  rq_init_comm_if_connected(9, "1")
  rq_init_comm_if_connected(2, "2")
  rq_init_comm_if_connected(3, "3")
  rq_init_comm_if_connected(4, "4")
  rq_print_connected_grippers()
  rq_gripper_communication_thread = run rq_gripper_communication()
  set_closed_norm(100.0, 1)
  set_open_norm(0.0, 1)
  set_closed_mm(0.0, 1)
  set_open_mm(50.0, 1)
  set_closed_norm(89.80392156862744, 2)
  set_open_norm(1.1764705882352942, 2)
  set_closed_mm(0.0, 2)
  set_open_mm(85.0, 2)
  set_closed_norm(100.0, 3)
  set_open_norm(0.0, 3)
  set_closed_mm(0.0, 3)
  set_open_mm(50.0, 3)
  set_closed_norm(100.0, 4)
  set_open_norm(0.0, 4)
  set_closed_mm(0.0, 4)
  set_open_mm(50.0, 4)
  rq_current_limit_enabled = False
  while(not rq_gripper_communication_thread_started):
      sleep(0.008)
  end
  # end: URCap Installation Node
  global Waypoint_1_p=p[.239154028168, -.112421187536, .388460805492, -2.190061121647, 2.239885105363, -.031522131746]
  global Waypoint_1_q=[0.08494941145181656, -1.356790379886963, -1.3501760959625244, 4.298311873073242, 1.5503448247909546, -12.457233563551696]
  global Waypoint_2_p=p[.353622143993, -.121329124968, .189938870353, -2.206384372041, 2.219086090555, -.015107570982]
  global Waypoint_2_q=[0.029603084549307823, -1.8911191425719203, -1.7472671270370483, 5.225752520352163, 1.5633039474487305, -12.537665781119856]
  global Waypoint_3_p=p[.353631843850, -.121307264267, .374404133955, -2.206378505151, 2.218976644385, -.015136018793]
  global Waypoint_3_q=[0.028919491916894913, -1.8426815472044886, -0.9176297783851624, 4.347720308894775, 1.5626927614212036, -12.531363688895496]
  global Waypoint_4_p=p[.353652148585, -.121293807225, .374372255201, -3.125989777988, .006696998981, .003111919112]
  global Waypoint_4_q=[0.02515784278512001, -1.855485578576559, -0.8932921886444092, 4.319008513087891, 1.5770167112350464, -14.107108545287538]
  global Waypoint_5_p=p[.363758828354, -.279187005666, .088904998077, -1.864461804969, .039872112715, .023313168997]
  global Waypoint_5_q=[-0.5345833937274378, -3.078116556207174, 0.038124863301412404, 3.5885044771381835, 2.5377118587493896, -15.200349044783998]
  global Waypoint_6_p=p[.362697799110, -.116842031967, .196258778113, -2.190025675108, 2.239949259838, -.031496290672]
  global Waypoint_6_q=[0.04410656914114952, -1.9051410160460414, -1.6960663795471191, 5.193034875183859, 1.5527570247650146, -12.506267488488945]
  global Waypoint_7_p=p[.362692894564, -.116852534259, .196244574783, -2.259726483789, -2.172286107875, .033806793645]
  global Waypoint_7_q=[0.04398636892437935, -1.9128123722472132, -1.6671544313430786, 5.131094622402944, 1.5524976253509521, -9.347179301569255]
  global Waypoint_8_p=p[.364841512775, -.116912589132, .188280404566, -3.140213348041, .061797284546, .022617550423]
  global Waypoint_8_q=[0.04088902473449707, -1.9356409511961878, -1.678733229637146, 5.171853232174673, 1.5633610486984253, -14.06320519445746]
  global Waypoint_9_p=p[.364848248729, -.116916737546, .353527898805, -3.140241647694, .061909886054, .022584279111]
  global Waypoint_9_q=[0.040220536291599274, -1.8723865948119105, -0.9687836766242981, 4.39864365636792, 1.5626797676086426, -14.057535123809267]
  global Waypoint_10_p=p[.360930807194, -.273182609942, .095849475862, -1.840638665045, .023655413076, -.007249116988]
  global Waypoint_10_q=[-0.5289800802813929, -2.9153500996031703, -0.2807917296886444, 3.7200543123432617, 2.5632033348083496, -15.246222686751771]
  global Waypoint_11_p=p[.358486190954, -.117341083615, .189882871874, -2.190038242218, 2.239881886121, -.031548557662]
  global Waypoint_11_q=[0.04321024566888809, -1.9022838077940882, -1.7338793277740479, 5.228053617268362, 1.5529053211212158, -12.50744832355717]
  global Waypoint_12_p=p[.358488238407, -.117335044807, .416524833090, -2.189975558032, 2.239914270517, -.031549652988]
  global Waypoint_12_q=[0.041965365409851074, -1.9908906422057093, -0.4767185151576996, 4.059401198024414, 1.5538296699523926, -12.499717981109413]
  global Waypoint_13_p=p[.358499834191, -.117338038000, .416498790970, -.024529661157, -3.133343015716, .032078362261]
  global Waypoint_13_q=[0.04467107728123665, -2.0224882564940394, -0.4105936884880066, 3.9957544046589355, 1.5432183742523193, -10.932522662470134]
  global Waypoint_14_p=p[.366071635210, -.114893443374, .213688173446, -.024436496176, -3.133440569951, .032084448400]
  global Waypoint_14_q=[0.05177054554224014, -1.8911673031248988, -1.61358642578125, 5.067582773953237, 1.5413740873336792, -10.9335692008231]
  while (True):
    $ 1 "Robot Program"
    $ 2 "MoveJ"
    $ 3 "Waypoint_1" "breakAfter"
    movej(get_inverse_kin(Waypoint_1_p, qnear=Waypoint_1_q), a=1.3962634015954636, v=1.0471975511965976)
    $ 4 "MoveJ"
    $ 5 "Waypoint_2" "breakAfter"
    movej(get_inverse_kin(Waypoint_2_p, qnear=Waypoint_2_q), a=1.3962634015954636, v=1.0471975511965976)
    # begin: URCap Program Node
    #   Source: Robotiq_Grippers, 1.8.11.21258, Robotiq Inc.
    #   Type: Gripper
    $ 6 "Gripper Close (2)"
    if not(gripper_connected[1]):
      popup("Gripper 2 must be connected to run this program.", "No connection", False, True, True)
    end
    if not(rq_is_gripper_activated("2")):
      popup("Gripper 2 is not activated. Go to Installation tab > Gripper to activate it and run the program again.", "Not activated", False, True, True)
    end
    rq_set_pos_spd_for(255, 0, 0, "2")
    rq_wait_pos_spe_for_request(255, 0, 0, "2")
    rq_go_to("2")
    rq_wait("2")
    # end: URCap Program Node
    $ 7 "MoveJ"
    $ 8 "Waypoint_3" "breakAfter"
    movej(get_inverse_kin(Waypoint_3_p, qnear=Waypoint_3_q), a=1.3962634015954636, v=1.0471975511965976)
    $ 9 "MoveJ"
    $ 10 "Waypoint_4" "breakAfter"
    movej(get_inverse_kin(Waypoint_4_p, qnear=Waypoint_4_q), a=1.3962634015954636, v=1.0471975511965976)
    $ 11 "MoveJ"
    $ 12 "Waypoint_5" "breakAfter"
    movej(get_inverse_kin(Waypoint_5_p, qnear=Waypoint_5_q), a=1.3962634015954636, v=1.0471975511965976)
    # begin: URCap Program Node
    #   Source: Robotiq_Grippers, 1.8.11.21258, Robotiq Inc.
    #   Type: Gripper
    $ 13 "Gripper Open (2)"
    if not(gripper_connected[1]):
      popup("Gripper 2 must be connected to run this program.", "No connection", False, True, True)
    end
    if not(rq_is_gripper_activated("2")):
      popup("Gripper 2 is not activated. Go to Installation tab > Gripper to activate it and run the program again.", "Not activated", False, True, True)
    end
    rq_set_pos_spd_for(0, 0, 0, "2")
    rq_wait_pos_spe_for_request(0, 0, 0, "2")
    rq_go_to("2")
    rq_wait("2")
    # end: URCap Program Node
    $ 14 "MoveJ"
    $ 15 "Waypoint_1" "breakAfter"
    movej(get_inverse_kin(Waypoint_1_p, qnear=Waypoint_1_q), a=1.3962634015954636, v=1.0471975511965976)
    $ 16 "MoveJ"
    $ 17 "Waypoint_6" "breakAfter"
    movej(get_inverse_kin(Waypoint_6_p, qnear=Waypoint_6_q), a=1.3962634015954636, v=1.0471975511965976)
    # begin: URCap Program Node
    #   Source: Robotiq_Grippers, 1.8.11.21258, Robotiq Inc.
    #   Type: Gripper
    $ 18 "Gripper Close (2)"
    if not(gripper_connected[1]):
      popup("Gripper 2 must be connected to run this program.", "No connection", False, True, True)
    end
    if not(rq_is_gripper_activated("2")):
      popup("Gripper 2 is not activated. Go to Installation tab > Gripper to activate it and run the program again.", "Not activated", False, True, True)
    end
    rq_set_pos_spd_for(255, 0, 0, "2")
    rq_wait_pos_spe_for_request(255, 0, 0, "2")
    rq_go_to("2")
    rq_wait("2")
    # end: URCap Program Node
    $ 19 "MoveJ"
    $ 20 "Waypoint_7" "breakAfter"
    movej(get_inverse_kin(Waypoint_7_p, qnear=Waypoint_7_q), a=1.3962634015954636, v=1.0471975511965976)
    # begin: URCap Program Node
    #   Source: Robotiq_Grippers, 1.8.11.21258, Robotiq Inc.
    #   Type: Gripper
    $ 21 "Gripper Open (2)"
    if not(gripper_connected[1]):
      popup("Gripper 2 must be connected to run this program.", "No connection", False, True, True)
    end
    if not(rq_is_gripper_activated("2")):
      popup("Gripper 2 is not activated. Go to Installation tab > Gripper to activate it and run the program again.", "Not activated", False, True, True)
    end
    rq_set_pos_spd_for(0, 0, 0, "2")
    rq_wait_pos_spe_for_request(0, 0, 0, "2")
    rq_go_to("2")
    rq_wait("2")
    # end: URCap Program Node
    $ 22 "MoveJ"
    $ 23 "Waypoint_1" "breakAfter"
    movej(get_inverse_kin(Waypoint_1_p, qnear=Waypoint_1_q), a=1.3962634015954636, v=1.0471975511965976)
    $ 24 "MoveJ"
    $ 25 "Waypoint_8" "breakAfter"
    movej(get_inverse_kin(Waypoint_8_p, qnear=Waypoint_8_q), a=1.3962634015954636, v=1.0471975511965976)
    # begin: URCap Program Node
    #   Source: Robotiq_Grippers, 1.8.11.21258, Robotiq Inc.
    #   Type: Gripper
    $ 26 "Gripper Close (2)"
    if not(gripper_connected[1]):
      popup("Gripper 2 must be connected to run this program.", "No connection", False, True, True)
    end
    if not(rq_is_gripper_activated("2")):
      popup("Gripper 2 is not activated. Go to Installation tab > Gripper to activate it and run the program again.", "Not activated", False, True, True)
    end
    rq_set_pos_spd_for(255, 0, 0, "2")
    rq_wait_pos_spe_for_request(255, 0, 0, "2")
    rq_go_to("2")
    rq_wait("2")
    # end: URCap Program Node
    $ 27 "MoveJ"
    $ 28 "Waypoint_9" "breakAfter"
    movej(get_inverse_kin(Waypoint_9_p, qnear=Waypoint_9_q), a=1.3962634015954636, v=1.0471975511965976)
    $ 29 "MoveJ"
    $ 30 "Waypoint_10" "breakAfter"
    movej(get_inverse_kin(Waypoint_10_p, qnear=Waypoint_10_q), a=1.3962634015954636, v=1.0471975511965976)
    # begin: URCap Program Node
    #   Source: Robotiq_Grippers, 1.8.11.21258, Robotiq Inc.
    #   Type: Gripper
    $ 31 "Gripper Open (2)"
    if not(gripper_connected[1]):
      popup("Gripper 2 must be connected to run this program.", "No connection", False, True, True)
    end
    if not(rq_is_gripper_activated("2")):
      popup("Gripper 2 is not activated. Go to Installation tab > Gripper to activate it and run the program again.", "Not activated", False, True, True)
    end
    rq_set_pos_spd_for(0, 0, 0, "2")
    rq_wait_pos_spe_for_request(0, 0, 0, "2")
    rq_go_to("2")
    rq_wait("2")
    # end: URCap Program Node
    $ 32 "MoveJ"
    $ 33 "Waypoint_1" "breakAfter"
    movej(get_inverse_kin(Waypoint_1_p, qnear=Waypoint_1_q), a=1.3962634015954636, v=1.0471975511965976)
    $ 34 "MoveJ"
    $ 35 "Waypoint_8" "breakAfter"
    movej(get_inverse_kin(Waypoint_8_p, qnear=Waypoint_8_q), a=1.3962634015954636, v=1.0471975511965976)
    # begin: URCap Program Node
    #   Source: Robotiq_Grippers, 1.8.11.21258, Robotiq Inc.
    #   Type: Gripper
    $ 36 "Gripper Close (2)"
    if not(gripper_connected[1]):
      popup("Gripper 2 must be connected to run this program.", "No connection", False, True, True)
    end
    if not(rq_is_gripper_activated("2")):
      popup("Gripper 2 is not activated. Go to Installation tab > Gripper to activate it and run the program again.", "Not activated", False, True, True)
    end
    rq_set_pos_spd_for(255, 0, 0, "2")
    rq_wait_pos_spe_for_request(255, 0, 0, "2")
    rq_go_to("2")
    rq_wait("2")
    # end: URCap Program Node
    $ 37 "MoveJ"
    $ 38 "Waypoint_9" "breakAfter"
    movej(get_inverse_kin(Waypoint_9_p, qnear=Waypoint_9_q), a=1.3962634015954636, v=1.0471975511965976)
    $ 39 "MoveJ"
    $ 40 "Waypoint_10" "breakAfter"
    movej(get_inverse_kin(Waypoint_10_p, qnear=Waypoint_10_q), a=1.3962634015954636, v=1.0471975511965976)
    # begin: URCap Program Node
    #   Source: Robotiq_Grippers, 1.8.11.21258, Robotiq Inc.
    #   Type: Gripper
    $ 41 "Gripper Open (2)"
    if not(gripper_connected[1]):
      popup("Gripper 2 must be connected to run this program.", "No connection", False, True, True)
    end
    if not(rq_is_gripper_activated("2")):
      popup("Gripper 2 is not activated. Go to Installation tab > Gripper to activate it and run the program again.", "Not activated", False, True, True)
    end
    rq_set_pos_spd_for(0, 0, 0, "2")
    rq_wait_pos_spe_for_request(0, 0, 0, "2")
    rq_go_to("2")
    rq_wait("2")
    # end: URCap Program Node
    $ 42 "MoveJ"
    $ 43 "Waypoint_1" "breakAfter"
    movej(get_inverse_kin(Waypoint_1_p, qnear=Waypoint_1_q), a=1.3962634015954636, v=1.0471975511965976)
    $ 44 "MoveJ"
    $ 45 "Waypoint_8" "breakAfter"
    movej(get_inverse_kin(Waypoint_8_p, qnear=Waypoint_8_q), a=1.3962634015954636, v=1.0471975511965976)
    # begin: URCap Program Node
    #   Source: Robotiq_Grippers, 1.8.11.21258, Robotiq Inc.
    #   Type: Gripper
    $ 46 "Gripper Close (2)"
    if not(gripper_connected[1]):
      popup("Gripper 2 must be connected to run this program.", "No connection", False, True, True)
    end
    if not(rq_is_gripper_activated("2")):
      popup("Gripper 2 is not activated. Go to Installation tab > Gripper to activate it and run the program again.", "Not activated", False, True, True)
    end
    rq_set_pos_spd_for(255, 0, 0, "2")
    rq_wait_pos_spe_for_request(255, 0, 0, "2")
    rq_go_to("2")
    rq_wait("2")
    # end: URCap Program Node
    $ 47 "MoveJ"
    $ 48 "Waypoint_9" "breakAfter"
    movej(get_inverse_kin(Waypoint_9_p, qnear=Waypoint_9_q), a=1.3962634015954636, v=1.0471975511965976)
    $ 49 "MoveJ"
    $ 50 "Waypoint_10" "breakAfter"
    movej(get_inverse_kin(Waypoint_10_p, qnear=Waypoint_10_q), a=1.3962634015954636, v=1.0471975511965976)
    # begin: URCap Program Node
    #   Source: Robotiq_Grippers, 1.8.11.21258, Robotiq Inc.
    #   Type: Gripper
    $ 51 "Gripper Open (2)"
    if not(gripper_connected[1]):
      popup("Gripper 2 must be connected to run this program.", "No connection", False, True, True)
    end
    if not(rq_is_gripper_activated("2")):
      popup("Gripper 2 is not activated. Go to Installation tab > Gripper to activate it and run the program again.", "Not activated", False, True, True)
    end
    rq_set_pos_spd_for(0, 0, 0, "2")
    rq_wait_pos_spe_for_request(0, 0, 0, "2")
    rq_go_to("2")
    rq_wait("2")
    # end: URCap Program Node
    $ 52 "MoveJ"
    $ 53 "Waypoint_1" "breakAfter"
    movej(get_inverse_kin(Waypoint_1_p, qnear=Waypoint_1_q), a=1.3962634015954636, v=1.0471975511965976)
    $ 54 "MoveJ"
    $ 55 "Waypoint_11" "breakAfter"
    movej(get_inverse_kin(Waypoint_11_p, qnear=Waypoint_11_q), a=1.3962634015954636, v=1.0471975511965976)
    # begin: URCap Program Node
    #   Source: Robotiq_Grippers, 1.8.11.21258, Robotiq Inc.
    #   Type: Gripper
    $ 56 "Gripper Close (2)"
    if not(gripper_connected[1]):
      popup("Gripper 2 must be connected to run this program.", "No connection", False, True, True)
    end
    if not(rq_is_gripper_activated("2")):
      popup("Gripper 2 is not activated. Go to Installation tab > Gripper to activate it and run the program again.", "Not activated", False, True, True)
    end
    rq_set_pos_spd_for(255, 0, 0, "2")
    rq_wait_pos_spe_for_request(255, 0, 0, "2")
    rq_go_to("2")
    rq_wait("2")
    # end: URCap Program Node
    $ 57 "MoveJ"
    $ 58 "Waypoint_12" "breakAfter"
    movej(get_inverse_kin(Waypoint_12_p, qnear=Waypoint_12_q), a=1.3962634015954636, v=1.0471975511965976)
    $ 59 "MoveJ"
    $ 60 "Waypoint_13" "breakAfter"
    movej(get_inverse_kin(Waypoint_13_p, qnear=Waypoint_13_q), a=1.3962634015954636, v=1.0471975511965976)
    $ 61 "MoveJ"
    $ 62 "Waypoint_14" "breakAfter"
    movej(get_inverse_kin(Waypoint_14_p, qnear=Waypoint_14_q), a=1.3962634015954636, v=1.0471975511965976)
    # begin: URCap Program Node
    #   Source: Robotiq_Grippers, 1.8.11.21258, Robotiq Inc.
    #   Type: Gripper
    $ 63 "Gripper Open (2)"
    if not(gripper_connected[1]):
      popup("Gripper 2 must be connected to run this program.", "No connection", False, True, True)
    end
    if not(rq_is_gripper_activated("2")):
      popup("Gripper 2 is not activated. Go to Installation tab > Gripper to activate it and run the program again.", "Not activated", False, True, True)
    end
    rq_set_pos_spd_for(0, 0, 0, "2")
    rq_wait_pos_spe_for_request(0, 0, 0, "2")
    rq_go_to("2")
    rq_wait("2")
    # end: URCap Program Node
    $ 64 "MoveJ"
    $ 65 "Waypoint_1" "breakAfter"
    movej(get_inverse_kin(Waypoint_1_p, qnear=Waypoint_1_q), a=1.3962634015954636, v=1.0471975511965976)
  end
end
